// SIMATIC STEP 7 (V5.x) project CovesCAO
// CPU: CPU 315-2 PN/DP
// station: Hardware
// station: P_ADR_BUS
// station: Line04
// program: Engineering ZE25 - Common Program (Engineering) for Lines 01 & 02

SYMBOL_TABLE
"DB_GlobalData"	DB 1	DB 1	// Database global data
"DB_Keys"	DB 3	DB 3	// DB_Keys
"DB_Horn"	DB 5	DB 5	// Database Faults Horn request
"DB_VisuPara"	DB 6	DB 6	// Data from/to Visualizaton Parameter
"DB_VisuFaults"	DB 9	DB 9	// Data from/to Visualization Faults
"DB_VisuFaultsPrio"	DB 10	DB 10
"DB_CommWM001"	DB 40	DB 40	// DB_CommWM001
"DB_CommWM009"	DB 41	DB 41	// DB_CommWM009
"DB_CommWM011"	DB 42	DB 42	// DB_CommWM011
"DB_CommM0001"	DB 45	DB 45	// ABB ACS880 RPBA-01 interface EU MainDrive
"DB_CommM1103"	DB 46	DB 46	// ABB ACS880 RPBA-01 interface DT Sidefeeder
"DB_CommM0101"	DB 47	DB 47	// ABB ACS880 RPBA-01 interface BE BDP Dosing
"DB_CommM0102"	DB 48	DB 48	// ABB ACS880 RPBA-01 interface GR Pelletizer
"IDB_FB0"	DB 100	FB 0	// Instance data block of FB0
"IDB_FB1"	DB 101	FB 1	// Instance data block of FB1
"IDB_FB3"	DB 103	FB 3	// Instance data block of FB3
"IDB_FB4"	DB 104	FB 4	// Instance data block of FB4
"IDB_FB5"	DB 105	FB 5	// Instance data block of FB5
"IDB_FB6"	DB 106	FB 6	// Instance data block of FB6
"IDB_FB10"	DB 110	FB 10	// Instance data block of FB10
"IDB_FB11"	DB 111	FB 11	// Instance data block of FB11
"IDB_FB12"	DB 112	FB 12	// Instance data block of FB12
"IDB_FB13"	DB 113	FB 13	// Instance data block of FB13
"IDB_FB14"	DB 114	FB 14	// Instance data block of FB14
"IDB_FB15"	DB 115	FB 15	// Instance data block of FB15
"IDB_FB16"	DB 116	FB 16	// Instance data block of FB16
"IDB_FB17"	DB 117	FB 17	// Instance data block of FB17
"IDB_FB27"	DB 127	FB 27	// Instance data block of FB27
"IDB_FB28"	DB 128	FB 28	// Instance data block of FB28
"IDB_FB29"	DB 129	FB 29	// Instance data block of FB29
"IDB_FB30"	DB 130	FB 30	// Instance data block of FB30
"IDB_FB37"	DB 137	FB 37	// Instance data block of FB37
"IDB_FB40"	DB 140	FB 40	// Instance data block of FB40
"IDB_FB41"	DB 141	FB 41	// Instance data block of FB41
"IDB_FB42"	DB 142	FB 42	// Instance data block of FB42
"IDB_FB43"	DB 143	FB 43	// Instance data block of FB43
"IDB_FB44"	DB 144	FB 44	// Instance data block of FB44
"IDB_FB45"	DB 145	FB 45	// Instance data block of FB45
"IDB_FB46"	DB 146	FB 46	// Instance data block of FB46
"IDB_FB48"	DB 148	FB 48	// Instance data block of FB48
"IDB_FB49"	DB 149	FB 49	// Instance data block of FB49
"IDB_FB60"	DB 160	FB 60	// Instance data block of FB60
"IDB_FB61"	DB 161	FB 61	// Instance data block of FB61
"IDB_FB62"	DB 162	FB 62	// Instance data block of FB62
"IDB_FB70"	DB 170	FB 70	// Instance data block of FB70
"IDB_FB71"	DB 171	FB 71	// Instance data block of FB71
"IDB_FB72"	DB 172	FB 72	// Instance data block of FB72
"IDB_FB73"	DB 173	FB 73	// Instance data block of FB73
"IDB_FB74"	DB 174	FB 74	// Instance data block of FB74
"IDB_FB75"	DB 175	FB 75	// Instance data block of FB75
"IDB_FB76"	DB 176	FB 76	// Instance data block of FB76
"IDB_FB78"	DB 178	FB 78	// Instance data block of FB78
"IDB_FB100"	DB 1100	FB 100	// Instance data block of FB100
"IDB_FB112"	DB 1112	FB 112	// Instance data block of FB112
"IDB_FB116"	DB 1116	FB 116	// Instance data block of FB116
"IDB_FB117"	DB 1117	FB 117	// Instance data block of FB117
"Gen_Global"	FB 0	FB 0	// General Global
"Gen_GlobSig"	FB 1	FB 1	// General Global Signals
"EPGlobal"	FB 2	FB 2	// EPGlobal
"DPSlaveDiag"	FB 3	FB 3	// DP-Slave Diagnose
"FaultPrioSearch"	FB 4	FB 4	// MRoe Fault Priority Search
"HWButtonsStatus"	FB 5	FB 5	// HWButtonsStatus
"OperatingModes"	FB 6	FB 6	// OperatingModes Production / Maintenance
"BE_Org_Dos"	FB 10	FB 10	// BE Organisation Dosing
"BE_BC001DischargeFlap"	FB 11	FB 11	// BE BC001 discharge flap
"BE_BC001HopperInPos"	FB 12	FB 12	// BE BC001 hopper in position
"BE_BC001HopperPipeConn"	FB 13	FB 13	// BE BC001 hopper pipe connected
"BE_BC009DischargeAid"	FB 14	FB 14	// BE BC009 hopper discharge aid
"BE_BC009 DischargeFlap"	FB 15	FB 15	// BE_BC009 DischargeFlap
"BE_BC009 HopperInPos"	FB 16	FB 16	// BE_BC009 Hopper In Position
"BE_BC009HopperPipeConn"	FB 17	FB 17	// BE_BC009Hopper Pipe Connected
"BE_PA013Dosing"	FB 27	FB 27	// BE_PA013 dosing
"BE_PID PA013 OB35"	FB 28	FB 28	// BE PID controller for flow and temperature PA013 (OB35)
"BE_PA013Temperatures"	FB 29	FB 29	// BE_PA013Temperatures
"BE_PA013PropValve"	FB 30	FB 30	// PA013 proportional valve
"DT_EA011 Sidefeeder"	FB 37	FB 37	// DT EA011 Sidefeeder
"EU_Org_Extruder"	FB 40	FB 40	// EU Organisation Extruder - U0020
"EU_MainDrive"	FB 41	FB 41	// EU Extruder Main Drive - U0031
"EU_CoolingUnit"	FB 42	FB 42	// EU Cooling Unit - U0011
"EU_Clutch"	FB 43	FB 43	// EU extruder clutch
"EU_DriveCooling"	FB 44	FB 44	// EU main drive cooling - U0032
"EU_PIDCoolWaterTemp OB35"	FB 45	FB 45	// EU PID controller cooling water temperature (OB35)
"EU_NitrogenValve"	FB 46	FB 46	// EU Nitrogen valve
"EU_MeltPressTemp"	FB 48	FB 48	// EU extruder melt pressure and temperature
"EU_VacuumUnit"	FB 49	FB 49	// EU Extruder Vacuum Unit - U0024
"EU_Org_Heating"	FB 60	FB 60	// EU Organisation Heating
"EU_HeatingZone1"	FB 61	FB 61	// EU extruder heating zone 1 (feed zone)
"EU_HeatingZones2-11 OB35"	FB 62	FB 62	// EU Extruder Heating Zones 2 - 11 (OB35)
"GR_Org_Pel"	FB 70	FB 70	// GR Organisation Pelletizer
"GR_WaterBath"	FB 71	FB 71	// GR water bath pump - U0021
"GR_Dewatering"	FB 72	FB 72	// GR drive fan strand dewatering - U0022
"GR_Classifier"	FB 73	FB 73	// GR Classifier
"GR_SafetyKey"	FB 74	FB 74	// GR safety key
"GR_Pelletizer"	FB 75	FB 75	// GR pelletizer - U0023
"GR_PIDWaterBath"	FB 76	FB 76	// GR Water bath
"GR_DownstTotalizer"	FB 78	FB 78	// GR_DownstTotalizer
"DT_Org_Dos"	FB 100	FB 100	// DT Organisation Dosierung
"DT_WM001"	FB 112	FB 112	// DT WM001Brabender
"DT_WM009"	FB 116	FB 116	// DT WM009 KTron
"DT_WM011"	FB 117	FB 117	// DT_WM011 K-Tron
"EPTimerOn"	FB 304	FB 304
"EPTimerOff"	FB 305	FB 305
"EPSetDateTime"	FB 307	FB 307	// Set Date and Time by UDT0
"EPFindMaxDINT"	FB 309	FB 309	// EPFindMaxDINT
"EPFilter"	FB 311	FB 311
"EPExPulsGen"	FB 317	FB 317	// EPExPulsGen
"EPThermIntegLoss"	FB 318	FB 318
"EPTempRamp"	FB 319	FB 319
"EPAverageVari"	FB 323	FB 323
"EPMotorN1FB"	FB 325	FB 325
"EPValveNC"	FB 336	FB 336	// EPValveNC
"EPFault"	FB 341	FB 341	// EPFault
"EPPreHeatTime"	FB 357	FB 357	// Extruder control and converting the pre heating time
"EPLevelSwitch"	FB 376	FB 376
"EPActValue"	FB 386	FB 386	// handling of ActREAL (modular SPS-datatype)
"EPRunTimeMeter"	FB 391	FB 391
"EPTotalPulse"	FB 392	FB 392
"EPToggle8"	FB 397	FB 397	// EPToggle8
"EPTcontZone"	FB 427	FB 427	// Extruder heating zone of tcont cp
"CONT_C"	FB 541	FB 541	// Continuous Control
"PULSEGEN"	FB 543	FB 543	// Pulse Generation
"TCONT_CP"	FB 558	FB 558	// temperature PID controller with pulse generator and self-tuning
"FCStatusWordsToVisu"	FB 603	FB 603	// FCStatusWordsToVisu
"BAYERDeviationAlmWarn"	FB 604	FB 604	// BAYERDeviationAlmWarn
"RF_RampAutoPush"	FB 615	FB 615	// Ramp value automatic to OP or inc/dec value by switches
"MR_TempZoneSimple"	FB 616	FB 616	// MR_TempZoneSimple
"CTBDHFlt"	FB 1000	FB 1000	// Störung für Dosierer
"CTKDLFlt"	FB 1001	FB 1001	// Dosierer K-Tron Detailstörungen
"EPGraph10Pos"	FB 1219	FB 1219
"EPRampOP_neu"	FB 1269	FB 1269	// EPRampOP_neu
"EPNomFilter"	FB 1270	FB 1270	// filtering of a nominal REAL value
"EPLocalMode"	FB 1282	FB 1282	// EPLocalMode
"EPTimerOn_neu"	FB 1304	FB 1304	// EPTimerOn_neu
"EPTimerOff_neu"	FB 1305	FB 1305	// EPTimerOff_neu
"EPAverageVari_Neu"	FB 1323	FB 1323
"EPMsg"	FB 1341	FB 1341
"EPSlaveDiagDP"	FB 1346	FB 1346	// Slave Diag DP
"EPToggel8_neu"	FB 1397	FB 1397	// EPToggel8_neu
"EP MS DataChange REAL"	FB 1501	FB 1501	// master - slave datachange handler for REAL values
"EP MS DataChange BOOL"	FB 1502	FB 1502	// master - slave datachange handler for boolean signals
"EP Comm ISC-CM Plus"	FB 1530	FB 1530	// Comm ISC-CM Plus
"EP ISC-CMp H Feeder"	FB 1535	FB 1535	// Brabender ISC CM plus H-type dosing feeder
"EP Comm K-Link KCM / SCM"	FB 1540	FB 1540	// Communication to K-Tron Smart K-Link KCM or SCM
"CT KCM LWF Feeder"	FB 1545	FB 1545	// K-Tron Smart K-Link KCM LWF-type dosing feeder
"GE_DT"	FC 12	FC 12	// Greater or Equal DT
"GT_DT"	FC 14	FC 14	// Greater Than DT
"SB_DT_TM"	FC 35	FC 35	// Subtract DT Time
"EPOperationMessage"	FC 301	FC 301	// Block vor one operation message
"EPNomLight"	FC 302	FC 302	// EPNomLight
"EPStartStop"	FC 307	FC 307	// EPStartStop
"EPToggle1"	FC 309	FC 309	// EPToggle1
"EPLimitAlarmReal"	FC 320	FC 320	// limit alarm generation
"EPAnyBitSet"	FC 349	FC 349	// EPAnyBitSet
"EPAnalogInReal"	FC 351	FC 351	// EPAnalogInReal
"EPAnalogOutReal"	FC 361	FC 361	// EPAnalogOutReal
"EPNominalComponent"	FC 365	FC 365	// nominal calculation of one dosing component
"EPMinuteImpulse"	FC 383	FC 383	// EPMinuteImpulse
"BAYERNomLightStartup"	FC 502	FC 502	// BAYERNomLight with Startup value handling
"EPNomLightDINT"	FC 503	FC 503	// EPNomLightDINT
"EPBAYER_TSD"	FC 505	FC 505	// EPBAYER Theoretical Strand Diameter
"EPBAYER_UPOStat"	FC 506	FC 506	// EPBAYER_UPOStat
"ClearBitsDelayed"	FC 510	FC 510	// ClearBitsDelayed
"EPGraphCalc"	FC 1219	FC 1219	// GraphCalc
"EPStatText"	FC 1300	FC 1300	// EP Status Text
"EPStat"	FC 1301	FC 1301	// common Status for Visu
"=PS230+SK02-1F4:14"	I 0.0	BOOL	// CIRCUIT BREAKER 230VAC O.K.
"=PS24+SK02-2F5:14"	I 0.1	BOOL	// CIRCUIT BREAKER 24VDC CONTROL VOLTAGE O.K.
"=PS24+SK02-3F5:14"	I 0.2	BOOL	// CIRCUIT BREAKER 24VDC LOAD VOLTAGE O.K.
"=ES+SK02-2K3:94"	I 0.3	BOOL	// EMERGENCY STOP RELAY ON
"=ES+CP01-3S1:34"	I 0.4	BOOL	// EMERGENCY STOP CONTROL PANEL EXTRUDER
"=ES+CP02-3S2:32"	I 0.5	BOOL	// NOT EMERGENCY STOP CONTROL PANEL PELLETIZER
"=ES+CP03-3S3:34"	I 0.6	BOOL	// EMERGENCY STOP EXTERNAL
"=ES+CP04-3S4:34"	I 0.7	BOOL	// EMERGENCY STOP EXTERNAL
"=EU04+CP01-1S1:14"	I 1.0	BOOL	// LAMP TEST
"=EU04+CP01-1S2:14"	I 1.1	BOOL	// HORN OFF
"=EU04+CP01-1S3:14"	I 1.2	BOOL	// H0008 AUXILIARY DRIVES START
"=EU04+CP01-1S4:12"	I 1.3	BOOL	// H0008 AUXILIARY DRIVES STOP
"=EU04+CP01-1S5:14"	I 1.4	BOOL	// H0001 EXTRUDER MAIN DRIVE START
"=EU04+CP01-1S6:12"	I 1.5	BOOL	// H0001 EXTRUDER MAIN DRIVE STOP
"=EU04+CP01-1S7:24"	I 1.6	BOOL	// H0009 EXTRUDER -
"=EU04+CP01-1S7:14"	I 1.7	BOOL	// H0009 EXTRUDER +
"=EU04+CP01-2S1:14"	I 2.0	BOOL	// H0101 FEEDING SYSTEM START
"=EU04+CP01-2S2:12"	I 2.1	BOOL	// H0101 FEEDING SYSTEM STOP
"=EU04+CP01-2S3:24"	I 2.2	BOOL	// H0102 FEEDING -
"=EU04+CP01-2S3:14"	I 2.3	BOOL	// H0102 FEEDING +
"+CP01-X4:14"	I 2.4	BOOL	// SPARE
"+CP01-X4:15"	I 2.5	BOOL	// SPARE
"+CP01-X4:16"	I 2.6	BOOL	// SPARE
"=ILUM+CP01-1E1:5"	I 2.7	BOOL	// COOLING UNIT CABINET +CP01 OK
"=GR04+CP02-1S4:24"	I 3.0	BOOL	// CUTTER SLOW
"=GR04+CP02-1S2:14"	I 3.1	BOOL	// CUTTER SRART
"=GR04+CP02-1S1:12"	I 3.2	BOOL	// CUTTER STOP
"=GR04+CP02-1S3:14"	I 3.3	BOOL	// LOCAL
"=GR04+CP02-1S3:24"	I 3.4	BOOL	// REMOTE
"=GR04+CP02-1S4:14"	I 3.5	BOOL	// CUTTER FAST
"=GR04+CP02-1S5:22"	I 3.6	BOOL	// FEED ROLL UP PRESSURE ON
"=GR04+CP02-1S5:14"	I 3.7	BOOL	// FEED ROLL UP PRESSURE OFF
"=BE04+BC001-G0014:4"	I 4.0	BOOL	// HOPPER BC001 IN POSITION
"=BE04+XB001-G0013:BK"	I 4.1	BOOL	// XB001 DISCHARGE PIPE CONNECTED
"=BE04+BC009-G0094:4"	I 4.2	BOOL	// HOPPER BC009 IN POSITION
"=DT04+WM001-H0101:14"	I 4.3	BOOL	// EXTRUDER DOSING WM001 MAINTENANCE SWITCH ON
"=BE04+XB009-G0093:BK"	I 4.4	BOOL	// XB009 DISCHARGE PIPE CONNECTED
"I4.5"	I 4.5	BOOL	// SPARE
"I4.6"	I 4.6	BOOL	// SPARE
"=DT04+WM011-M1101:J5:5"	I 4.7	BOOL	// DOSING UNIT WM011 REFILL
"=DT04+WM011-H1101:6"	I 5.0	BOOL	// DOSING UNIT WM011 MAINTENANCE SWITCH ON
"=DT04+WM009-M0901:J5:5"	I 5.1	BOOL	// DOSING UNIT WM009 REFILL
"=DT04+WM009-H0901:6"	I 5.2	BOOL	// DOSING UNIT WM009 MAINTENANCE SWITCH ON
"=ES+SK02-2K1:X2:Y32"	I 5.3	BOOL	// EMERGENCY STOP OK
"=ES+CP01-1S1:14"	I 5.4	BOOL	// LOAD VOLTAGE ON
"=DT04+WM009-G0901:WH"	I 5.5	BOOL	// DOSING UNIT WM009 SAFETY SWITCH
"I5.6"	I 5.6	BOOL	// SPARE
"I5.7"	I 5.7	BOOL	// SPARE
"I8.0"	I 8.0	BOOL	// SPARE
"I8.1"	I 8.1	BOOL	// SPARE
"=EU04+GA001-G0001:BK"	I 8.2	BOOL	// CLUTCH CONTROL
"I8.3"	I 8.3	BOOL	// SPARE
"I8.4"	I 8.4	BOOL	// SPARE
"I8.5"	I 8.5	BOOL	// SPARE
"=EU04+SK02-8Q1:14"	I 8.6	BOOL	// PUMP TEMPERING UNIT EXTRUDER MOTOR PROTECT. O.K.
"=EU04+PA001-H0011:14"	I 8.7	BOOL	// PUMP TEMPERING UNIT MAINTENANCE SWITCH ON
"=EU04+BA001-L0011:BK"	I 10.0	BOOL	// COOLING WATER HIGH
"=EU04+BA001-L0011:GY"	I 10.1	BOOL	// COOLING WATER NOT LOW
"+SK02-X4:97"	I 10.2	BOOL	// SPARE
"=EU04+SK02-40K1:X2:Y32"	I 10.3	BOOL	// EXTRUDER SAFETY SWITCH OK
"=EU04+GA001-G0002:8"	I 10.4	BOOL	// SAFETY SWITCH OF CONNECTION PART COVER LEFT
"=EU04+GA001-G0003:8"	I 10.5	BOOL	// SAFETY SWITCH OF CONNECTION PART COVER RIGHT
"=EU04+GA001-G0004:8"	I 10.6	BOOL	// SAFETY SWITCH OF COUPLING COVER
"=EU04+GA001-G0005:8"	I 10.7	BOOL	// SAFETY SWITCH HOPPER COVER
"=EU04+GA001-F0041:4"	I 11.0	BOOL	// EXTRUDER NITROGEN FLOW SWITCHING POINT A
"=EU04+GA001-F0041:2"	I 11.1	BOOL	// EXTRUDER NITROGEN FLOW SWITCHING POINT B
"I11.2"	I 11.2	BOOL	// SPARE
"I11.3"	I 11.3	BOOL	// SPARE
"I11.4"	I 11.4	BOOL	// SPARE
"I11.5"	I 11.5	BOOL	// SPARE
"I11.6"	I 11.6	BOOL	// SPARE
"I11.7"	I 11.7	BOOL	// SPARE
"=EU04+SK02-13A1:2"	I 32.0	BOOL	// EXTRUDER ZONE 2 CURRENT CONTROL O.K.
"=EU04+SK02-15A1:2"	I 32.1	BOOL	// EXTRUDER ZONE 3 CURRENT CONTROL O.K.
"=EU04+SK02-17A1:2"	I 32.2	BOOL	// EXTRUDER ZONE 4 CURRENT CONTROL O.K.
"=EU04+SK02-19A1:2"	I 32.3	BOOL	// EXTRUDER ZONE 5 CURRENT CONTROL O.K.
"=EU04+SK02-21A1:2"	I 32.4	BOOL	// EXTRUDER ZONE 6 CURRENT CONTROL O.K.
"=EU04+SK02-23A1:2"	I 32.5	BOOL	// EXTRUDER ZONE 7 CURRENT CONTROL O.K.
"=EU04+SK02-25A1:2"	I 32.6	BOOL	// EXTRUDER ZONE 8 CURRENT CONTROL O.K.
"=DT04+EA011-H1103:14"	I 32.7	BOOL	// SIDE FEEDER MAINTENANCE SWITCH ON
"=EU04+SK02-29A1:2"	I 33.0	BOOL	// EXTRUDER ZONE 10 CURRENT CONTROL O.K.
"=DT04+EA011-H1104:14"	I 33.1	BOOL	// SIDE FEEDER VACUUMPUMP ON
"=EU04+SK02-32K1:X6:OU2"	I 33.2	BOOL	// EXTRUDER MELT PRESSURE NOT MAX MAX
"=EU04+SK02-32K1:X6:OU1"	I 33.3	BOOL	// DIFFERENTIAL PRESSURE P1.1 <--> P1.2 MAX MAX
"=EU04+SK02-33K1:X6:OU1"	I 33.4	BOOL	// EXTRUDER ZONE 8 MELT PRESSURE MAX. MAX.
"=DT04+SK02-11Q1:14"	I 33.5	BOOL	// SIDE FEEDER VACUUMPUMP MOTOR PROTECT. O.K.
"=EU04+SK02-31A1:2"	I 33.6	BOOL	// EXTRUDER ZONE 11 CURRENT CONTROL O.K.
"I33.7"	I 33.7	BOOL	// SPARE
"=EU04+SK01-10T1:8"	I 140.0	BOOL	// VACUUM UNIT SEPARATOR NOT EMPTY
"=BE04+SK01-4Q1:14"	I 140.1	BOOL	// PA013 PUMP DRIVE MOTOR PROTECTION OK
"=BE04+PA013-H0101:14"	I 140.2	BOOL	// PUMP DRIVE PA013 MAINTENANCE SWITCH ON
"=BE04+SK01-8A1:12"	I 140.3	BOOL	// PA013 HEATER PUMP ZONE 2 CURRENT CONTROL O.K.
"=BE04+PA013-P0101:2"	I 140.4	BOOL	// PA013 PRESSURE >MIN
"I140.5"	I 140.5	BOOL	// SPARE
"=BE04+PA013-G0102:2"	I 140.6	BOOL	// PA013 GATE VALVE TO EXTRUDER OPEN
"=BE04+PA013-G0102:3"	I 140.7	BOOL	// PA013 GATE VALVE TO EXTRUDER CLOSED
"=BE04+PA013-G0101:2"	I 141.0	BOOL	// PA013 GATE VALVE RETURN FLOW OPENED
"=BE04+PA013-G0101:3"	I 141.1	BOOL	// PA013 GATE VALVE RETURN FLOW CLOSED
"=GR04+SK01-21Q1:14"	I 141.2	BOOL	// CLASSIFIER VIBRATOR MOTOR PROTECTION OK
"=EU04+SK01-11T1:12"	I 141.3	BOOL	// VACUUM UNIT SEPARATOR TEMPERATURE WARNING
"=GR04+SK01-13K1:Y32"	I 141.4	BOOL	// PELLETIZER NOT RUNNING
"=GR04+SK01-13K1:Y35"	I 141.5	BOOL	// PELLETIZER FAULT
"=EU04+GM001-H0001:14"	I 141.6	BOOL	// EXTRUDER DRIVE MAINTENANCE SWITCH ON
"=GR04+SK01-11Q1:14"	I 141.7	BOOL	// PELLETIZER DRIVE MOTOR PROTECTION OK
"=EU04+VP001-H0201:14"	I 142.0	BOOL	// VACUUM PUMP EXTRUDER MAINTENANCE SWITCH ON
"=EU04+SK01-8Q1:14"	I 142.1	BOOL	// VACUUM PUMP EXTRUDER MOTOR PROTECT. O.K.
"=GR04+PA001-H0201:14"	I 142.2	BOOL	// PUMP WATER BATH MAINTENANCE SWITCH ON
"I142.3"	I 142.3	BOOL	// SPARE
"I142.4"	I 142.4	BOOL	// SPARE
"=GR04+SK01-11Q2:14"	I 142.5	BOOL	// PELLETIZER DRIVE MOTOR CONTACTOR ON FEEDBACK MONITORING
"=ILUM+SK01-3E1:X1"	I 142.6	BOOL	// AIR CONDITIONER NO FAULT
"=GR04+ZA001-G0030:5"	I 142.7	BOOL	// SAFETY DOOR CLOSED
"=GR04+SK01-1Q1:14"	I 143.0	BOOL	// PUMP WATER BATH MOTOR PROTECT. O.K.
"I143.1"	I 143.1	BOOL	// SPARE
"I143.2"	I 143.2	BOOL	// SPARE
"=GR04+SK01-15K1:X2:Y32"	I 143.3	BOOL	// PELLETIZER KEY PLUGGED
"=ML04+PM001-SE-K1"	I 143.4	BOOL	// PACKING MACHINE RUNNING
"=ML04+PM001-SE-K2"	I 143.5	BOOL	// PACKING MACHINE FAULT
"=ML04+PM001-SE-K3"	I 143.6	BOOL	// PACKING MACHINE CONVEYOR RUNNING
"=ML04+PM001-SE-K4"	I 143.7	BOOL	// PACKING MACHINE BAG COUNTER
"=EU04+VP001-P0083:4"	I 144.0	BOOL	// VACUUM UNIT PRESSURE INDICATOR
"=EU04+SK01-12T1:21"	I 144.1	BOOL	// VACUUM UNIT FLOW SWITCH MIN
"=EU04+SK01-12T1:17"	I 144.2	BOOL	// VACUUM UNIT FLOW SWITCH FAULT
"=EU04+SK01-7Q1:14"	I 144.3	BOOL	// EXTRUDER FREMDBELÜFTUNG MOTOR PROTECT. O.K.
"+SK01-X7:37"	I 144.4	BOOL	// SPARE
"=DT04+SK01-1Q1:14"	I 144.5	BOOL	// SIDE FEEDER MOTOR PROTECT. O.K.
"+SK01-X7:38"	I 144.6	BOOL	// SPARE
"=EU04+GM001-H0002:14"	I 144.7	BOOL	// EXTRUDER FREMDBELÜFTUNG MAINTENANCE SWITCH ON
"Clock10000mHz"	M 0.0	BOOL	// clock signal 10Hz / 100ms
"Clock5000mHz"	M 0.1	BOOL	// clock signal 5Hz / 200ms
"Clock2500mHz"	M 0.2	BOOL	// clock signal 2,5Hz / 400ms
"Clock2000mHz"	M 0.3	BOOL	// clock signal 2Hz / 500ms
"Clock1250mHz"	M 0.4	BOOL	// clock signal 1,25Hz / 800ms
"Clock1000mHz"	M 0.5	BOOL	// clock signal 1Hz / 1s
"Clock625mHz"	M 0.6	BOOL	// clock signal 0,625Hz / 1,6s
"Clock500mHz"	M 0.7	BOOL	// clock signal 0,5Hz / 2s
"Impulse100ms"	M 1.0	BOOL	// impulse signal each 100ms
"Impulse200ms"	M 1.1	BOOL	// impulse signal each 200ms
"Impulse400ms"	M 1.2	BOOL	// impulse signal each 400ms
"Impulse500ms"	M 1.3	BOOL	// impulse signal each 500ms
"Impulse800ms"	M 1.4	BOOL	// impulse signal each 800ms
"Impulse1000ms"	M 1.5	BOOL	// impulse signal each 1000ms
"Impulse1600ms"	M 1.6	BOOL	// impulse signal each 1600ms
"Impulse2000ms"	M 1.7	BOOL	// impulse signal each 2000ms
"StartUpPLC"	M 2.0	BOOL	// start up signal, set in OB100/OB101/OB102, reset at end of program
"BatteryFault"	M 2.1	BOOL	// battery fault, set in OB81
"ControlVoltageOn"	M 2.2	BOOL	// control voltage on signal
"ControlVoltageOnDel"	M 2.3	BOOL	// control voltage on delayed signal
"LoadVoltageOn"	M 2.4	BOOL	// load voltage on signal extruder
"LoadVoltageOnDel"	M 2.5	BOOL	// load voltage on delayed signal extruder
"FaultAck"	M 2.6	BOOL	// fault acknowledge signal
"FaultAckExt"	M 2.7	BOOL	// fault acknowledge extended signal
"Impulse1min"	M 3.0	BOOL	// impulse signal each 1min
"LampTest"	M 3.1	BOOL	// extendet signal for lamp test
"BlockFault"	M 3.2	BOOL	// block fault signal
"HornAck"	M 3.3	BOOL	// horn acknowledge signal
"HornAckExt"	M 3.4	BOOL	// horn acknowledge extended signal
"ContrVoltageOnDel_Block"	M 3.5	BOOL	// block fault if control voltage is missing
"FaultAckOB35"	M 3.6	BOOL	// fault acknowledge signal for OB35
"HornAckOB35"	M 3.7	BOOL	// horn acknowledge signal for OB35
"LoadVoltageOnDel_Block"	M 4.0	BOOL	// block fault if load voltage is missing
"StartUpPLC_OB35"	M 4.4	BOOL	// start up signal for OB35, set in OB100/OB101/OB102, reset at end of OB35
"FaultOB80"	M 6.0	BOOL	// Fault: OB 80 called, cycle time error
"FaultOB81"	M 6.1	BOOL	// Fault: OB 81 called, power supply error
"FaultOB82"	M 6.2	BOOL	// Fault: OB 82 called, I/O point error 1
"FaultOB83"	M 6.3	BOOL	// Fault: OB 83 called, I/O point error 2
"FaultOB84"	M 6.4	BOOL	// Fault: OB 84 called, cpu error
"FaultOB85"	M 6.5	BOOL	// Fault: OB 85 called, OB not loaded
"FaultOB86"	M 6.6	BOOL	// Fault: OB 86 called, rack fault
"FaultOB87"	M 6.7	BOOL	// Fault: OB 87 called, communication fault
"FaultOB88"	M 7.0	BOOL	// Fault: OB 88 called, breakup error
"FaultOB121"	M 7.1	BOOL	// Fault: OB121 called, programming error
"FaultOB122"	M 7.2	BOOL	// Fault: OB122 called, module access error
"Simulation"	M 8.0	BOOL	// request start simulation [1=requested]
"IB_0"	M 10.0	BOOL	// commissioning & test always FALSE
"IB_1"	M 10.1	BOOL	// commissioning & test always TRUE
"IB_DummyOut"	M 10.2	BOOL	// commissioning & test for dummy outputs
"Alarm_Prio1"	M 100.0	BOOL	// Alarm with Priority 1 - safety alarm
"Alarm_Prio2"	M 100.1	BOOL	// Alarm with Priority 2 - process related alarm with interlock
"Alarm_Prio3"	M 100.2	BOOL	// Alarm with Priority 3 - process related alarm without interlock
"Alarm_Prio4"	M 100.3	BOOL	// Alarm with Priority 4 - event
"Alarm_Prio5"	M 100.4	BOOL	// Alarm with Priority 5 - system alarm
"FlagImpCoolDownOff"	M 110.2	BOOL	// Flag Impuls CoolDown Function Off
"ImpPA013PelletizerOff"	M 110.5	BOOL	// Impuls Pelletizer delayed off after PA013 Stop
"FlagImpPA013PelletOff"	M 111.5	BOOL	// Flag Impuls Pelletizer delayed off after PA013 Stop
"ClockByte"	MB 0	BYTE	// byte for clock signals
"ImpulseByte"	MB 1	BYTE	// byte for impulses
"MD10"	MD 10	REAL	// commissioning & test
"CycleExecution"	OB 1	OB 1	// CycleExecution
"CYC_INT5"	OB 35	OB 35	// Cyclic Interrupt 3
"CYCL_FLT"	OB 80	OB 80	// Cycle Time Fault
"I/O_FLT1"	OB 82	OB 82	// I/O Point Fault 1
"I/O_FLT2"	OB 83	OB 83	// I/O Point Fault 2
"OBNL_FLT"	OB 85	OB 85	// OB Not Loaded Fault
"RACK_FLT"	OB 86	OB 86	// Loss of Rack Fault
"COMM_FLT"	OB 87	OB 87	// Communication Fault
"EPCompleteRestart"	OB 100	OB 100	// EPCompleteRestart
"PROG_ERR"	OB 121	OB 121	// Programming Error
"MOD_ERR"	OB 122	OB 122	// Module Access Error
"=EU04+EA001-T0003:Fe"	PIW 320	INT	// EXTRUDER FEED ZONE TEMPERATURE
"=EU04+EA001-T0021:Fe"	PIW 322	INT	// EXTRUDER ZONE 2 TEMPERATURE
"=EU04+EA001-T0031:Fe"	PIW 324	INT	// EXTRUDER ZONE 3 TEMPERATURE
"=EU04+EA001-T0041:Fe"	PIW 326	INT	// EXTRUDER ZONE 4 TEMPERATURE
"=EU04+EA001-T0051:Fe"	PIW 328	INT	// EXTRUDER ZONE 5 TEMPERATURE
"=EU04+EA001-T0061:Fe"	PIW 330	INT	// EXTRUDER ZONE 6 TEMPERATURE
"=EU04+EA001-T0071:Fe"	PIW 332	INT	// EXTRUDER ZONE 7 TEMPERATURE
"=EU04+EA001-T0081:Fe"	PIW 334	INT	// EXTRUDER ZONE 8 TEMPERATURE
"PIW336"	PIW 336	INT	// SPARE
"PIW338"	PIW 338	INT	// SPARE
"=EU04+EA001-T0101:Fe"	PIW 340	INT	// EXTRUDER ZONE 10 TEMPERATURE
"=EU04+EA001-T0102:Fe"	PIW 342	INT	// EXTRUDER ZONE 11 TEMPERATURE
"=EU04+EA001-T0112:Fe"	PIW 344	INT	// EXTRUDER MELT TEMPERATURE
"=EU04+PA001-T0011:Fe"	PIW 346	INT	// TEMPERATURE COOLING WATER TEMPERING UNIT
"PIW348"	PIW 348	INT	// SPARE
"PIW350"	PIW 350	INT	// SPARE
"=EU04+SK02-32K1:X4:1"	PIW 352	INT	// MELT PRESSURE P1.1 ACTUAL VALUE
"=EU04+SK02-32K1:X4:2"	PIW 354	INT	// MELT PRESSURE P1.2 ACTUAL VALUE
"=EU04+SK02-33K1:X4:1"	PIW 356	INT	// EXTRUDER MELT PRESSURE ACTUAL VALUE
"=EU04+GA001-F0041:5"	PIW 358	INT	// EXTRUDER NITROGEN FLOW ACTUAL VALUE
"=BE04+BC001-Y0012:9"	PIW 360	INT	// DISCHARGE FLAP BC001 OPEN ACTUAL VALUE
"PIW362"	PIW 362	INT	// SPARE
"=BE04+BC009-Y0092:9"	PIW 364	INT	// DISCHARGE FLAP BC009 OPEN ACTUAL VALUE
"PIW366"	PIW 366	INT	// SPARE
"PIW368"	PIW 368	INT	// SPARE
"PIW370"	PIW 370	INT	// SPARE
"PIW372"	PIW 372	INT	// SPARE
"PIW374"	PIW 374	INT	// SPARE
"=BE04+PA013-T0313:1"	PIW 380	INT	// PA013 TEMPERATURE ZONE 1 BEVORE PUMPE
"=BE04+PA013-T0314:1"	PIW 382	INT	// PA013 TEMPERATURE ZONE 3 PUMP
"=BE04+PA013-T0315:1"	PIW 384	INT	// PA013 TEMPERATURE ZONE 4 AFTER PUMP
"=BE04+PA013-T0316:1"	PIW 386	INT	// PA013 TEMPERATURE ZONE 5 ANSCHLUSSSTÜCK EXTRUDER
"=BE04+PA013-T0102:1"	PIW 388	INT	// PA013 TEMPERATURE PUMP ZONE 2
"=GR04+FB001-T0042:1"	PIW 390	INT	// CLASSIFIER FB001 TEMPERATURE PRODUCT
"=BE04+PA013-T0107:1"	PIW 392	INT	// PA013 TEMPERATURE PRODUCT
"PIW394"	PIW 394	INT	// SPARE
"+SK01-X7:39"	PIW 396	INT	// SPARE
"=EU04+VP001-P0083:2"	PIW 398	INT	// VACUUM UNIT ACTUAL PRESSURE
"=GR04+WX001-T0011:+"	PIW 400	INT	// RECIRCLE WATER SUPPLY TEMPERATURE
"=GR04+WX001-T0012:+"	PIW 402	INT	// RECIRCLE WATER RETURE TEMPERATURE
"=EU04+SK01-11T1:7"	PIW 404	INT	// VACUUM UNIT SEPARATOR TEMPERATURE ACTUAL VALUE
"=GR04+FA001-P0101:1"	PIW 406	INT	// COOLING WATER PRESSURE ACTUAL VALUE
"=BE04+PA013-F0101:26"	PIW 408	INT	// PA013 FLOW MEASURING ACTUAL VALUE
"=BE04+PA013-P0102:1"	PIW 410	INT	// PA013 BDP DOSING PRESSURE ACTUAL VALUE
"=BE04+BC001-Y0012:1"	PQW 320	INT	// DISCHARGE FLAP BC001 OPEN NOMINAL VALUE
"=BE04+BC009-Y0092:1"	PQW 322	INT	// DISCHARGE FLAP BC009 OPEN NOMINAL VALUE
"PQW324"	PQW 324	INT	// SPARE
"PQW326"	PQW 326	INT	// SPARE
"=BE04+PA013-Y1320:11"	PQW 380	INT	// PA013 PROPORTIONAL VALVE
"=GR04+WA001-Y0011:11"	PQW 382	INT	// COOLING WATER RETURN VALVE
"PQW336"	PQW 384	INT	// SPARE
"PQW338"	PQW 386	INT	// SPARE
"=EU04+CP01-3P2:X1"	Q 0.0	BOOL	// LOAD VOLTAGE ON
"=EU04+CP01-3P3:X1"	Q 0.1	BOOL	// X0008 AUXILIARY DRIVES ON
"=EU04+CP01-3P4:X1"	Q 0.2	BOOL	// X0001 EXTRUDER MAIN DRIVE ON
"=EU04+CP01-3P5:X1"	Q 0.3	BOOL	// X0101 FEEDING SYSTEM ON
"+CP01-X4:25"	Q 0.4	BOOL	// SPARE
"+CP01-X4:26"	Q 0.5	BOOL	// SPARE
"+CP01-X4:27"	Q 0.6	BOOL	// SPARE
"+CP01-X4:28"	Q 0.7	BOOL	// SPARE
"Q1.0"	Q 1.0	BOOL	// SPARE
"Q1.1"	Q 1.1	BOOL	// SPARE
"Q1.2"	Q 1.2	BOOL	// SPARE
"=EU04+SK02-40K2:A1"	Q 1.3	BOOL	// EXTRUDER SAFETY SWITCH RESET
"Q1.4"	Q 1.4	BOOL	// SPARE
"=GR04+CP02-2P3:X1"	Q 1.5	BOOL	// CUTTER INTERLOCKING SYSTEM RELEASE
"=GR04+CP02-2P1:X1"	Q 1.6	BOOL	// CUTTER ON
"=GR04+CP02-2P2:X1"	Q 1.7	BOOL	// FEED ROLL UP PRESSURE OFF
"=DT04+WM001-2A2:68"	Q 2.0	BOOL	// DOSING UNIT WM001 RELEASE
"=DT04+SK02-8K1:A1"	Q 2.1	BOOL	// DOSING UNIT WM011 INTERLOCKING ON
"=DT04+SK02-6K1:A1"	Q 2.2	BOOL	// DOSING UNIT WM009 INTERLOCKING ON
"=ES+SK02-1K1:A1"	Q 2.3	BOOL	// EMERGENCY STOP RESET
"Q2.4"	Q 2.4	BOOL	// SPARE
"Q2.5"	Q 2.5	BOOL	// SPARE
"Q2.6"	Q 2.6	BOOL	// SPARE
"Q2.7"	Q 2.7	BOOL	// SPARE
"Q 3.0"	Q 3.0	BOOL	// spare
"=EU04+GA001-Y0012"	Q 3.1	BOOL	// COOLING WATER EXTRUDER GEAR BOX OPEN
"=EU04+SK02-8Q2:A1"	Q 3.2	BOOL	// PUMP TEMPERING UNIT EXTRUDER ON
"=EU04+WA001-Y0012:A1"	Q 3.3	BOOL	// COOLING WATER TEMPERING UNIT OPEN
"Q3.4"	Q 3.4	BOOL	// SPARE
"Q3.5"	Q 3.5	BOOL	// SPARE
"Q3.6"	Q 3.6	BOOL	// SPARE
"=EU04+BA001-Y0011:A1"	Q 3.7	BOOL	// INLET COOLING WATER TEMPERING UNIT OPEN
"=EU04+SK02-13V1:A1"	Q 32.0	BOOL	// EXTRUDER ZONE 2 HEATING ON
"=EU04+SK02-15V1:A1"	Q 32.1	BOOL	// EXTRUDER ZONE 3 HEATING ON
"=EU04+SK02-17V1:A1"	Q 32.2	BOOL	// EXTRUDER ZONE 4 HEATING ON
"=EU04+SK02-19V1:A1"	Q 32.3	BOOL	// EXTRUDER ZONE 5 HEATING ON
"=EU04+SK02-21V1:A1"	Q 32.4	BOOL	// EXTRUDER ZONE 6 HEATING ON
"=EU04+SK02-23V1:A1"	Q 32.5	BOOL	// EXTRUDER ZONE 7 HEATING ON
"=EU04+SK02-25V1:A1"	Q 32.6	BOOL	// EXTRUDER ZONE 8 HEATING ON
"=EU04+GA001-Y0045:1"	Q 32.7	BOOL	// EXTRUDER NITROGEN VALVE
"=EU04+SK02-29V1:A1"	Q 33.0	BOOL	// EXTRUDER ZONE 10 HEATING ON
"=EU04+SK02-31V1:A1"	Q 33.1	BOOL	// EXTRUDER ZONE 11 HEATING ON
"Q33.2"	Q 33.2	BOOL	// SPARE
"=BE04+BC009-Y0093:1"	Q 33.3	BOOL	// HOPPER BC009 KNOCKER ON
"=DT04+VP011-Y1101:1"	Q 33.4	BOOL	// SIDE FEEDER VACUUMPUMP AIR PURGE VALVE
"=DT04+VP011-Y1102:1"	Q 33.5	BOOL	// SIDE FEEDER VACUUMPUMP SUCTION VALVE
"=DT04+SK02-11Q2:A1"	Q 33.6	BOOL	// SIDE FEEDER VACUUMPUMP ON
"Q33.7"	Q 33.7	BOOL	// SPARE
"=EU04+SK02-32K1:X3:IN1"	Q 34.0	BOOL	// EXTRUDER MELT PRESSURE CALIBRATION
"=EU04+SK02-32K1:X3:IN3"	Q 34.1	BOOL	// EXTRUDER MELT PRESSURE RESET FAULT
"=EU04+SK02-33K1:X3:IN3"	Q 34.2	BOOL	// EXTRUDER MELT PRESSURE RESET FAULT
"=EU04+SK02-33K1:X3:IN1"	Q 34.3	BOOL	// EXTRUDER MELT PRESSURE CALIBRATION
"Q34.4"	Q 34.4	BOOL	// SPARE
"Q34.5"	Q 34.5	BOOL	// SPARE
"Q34.6"	Q 34.6	BOOL	// SPARE
"Q34.7"	Q 34.7	BOOL	// SPARE
"=EU04+EA001-Y0021:1"	Q 35.0	BOOL	// EXTRUDER ZONE 2 COOLING ON
"=EU04+EA001-Y0031:1"	Q 35.1	BOOL	// EXTRUDER ZONE 3 COOLING ON
"=EU04+EA001-Y0041:1"	Q 35.2	BOOL	// EXTRUDER ZONE 4 COOLING ON
"=EU04+EA001-Y0051:1"	Q 35.3	BOOL	// EXTRUDER ZONE 5 COOLING ON
"=EU04+EA001-Y0061:1"	Q 36.0	BOOL	// EXTRUDER ZONE 6 COOLING ON
"=EU04+EA001-Y0071:1"	Q 36.1	BOOL	// EXTRUDER ZONE 7 COOLING ON
"=EU04+EA001-Y0081:1"	Q 36.2	BOOL	// EXTRUDER ZONE 8 COOLING ON
"Q36.3"	Q 36.3	BOOL	// SPARE
"=GI+SK01-1P1:+"	Q 40.0	BOOL	// OPERATING HOURS COUNTER
"=GI+SK01-1K1:A1"	Q 40.1	BOOL	// SIGNAL HORN FAULT INDICATION
"=GI+SK01-2P1:2"	Q 40.2	BOOL	// SIGNAL LAMP RD
"=GI+SK01-2P1:1"	Q 40.3	BOOL	// SIGNAL LAMP YE
"=GI+SK01-2P1:3"	Q 40.4	BOOL	// SPARE
"=GR04+SK01-11Q2:A1"	Q 40.5	BOOL	// PELLETIZER DRIVE MOTOR CONTACTOR ON
"=GR04+SK01-15K2:A1"	Q 40.6	BOOL	// PELLETIZER SAFETY RELAY RESET
"Q40.7"	Q 40.7	BOOL	// SPARE
"Q41.0"	Q 41.0	BOOL	// SPARE
"Q41.1"	Q 41.1	BOOL	// SPARE
"=BE04+SK01-8A1:IN"	Q 41.2	BOOL	// PA013 HEATER PUMP ZONE 2 HEATING ON
"=BE04+PA013-G0102:5"	Q 41.3	BOOL	// PA013 GATE VALVE TO EXTRUDER OPEN
"=BE04+PA013-G0101:5"	Q 41.4	BOOL	// PA013 GATE VALVE RETURN FLOW OPEN
"=GR04+SK01-13K1:RESET"	Q 41.5	BOOL	// PELLETIZER RESET
"=GR04+ZA001-Y0102:1"	Q 41.6	BOOL	// FEED ROLL UP PRESSURE ON
"Q41.7"	Q 41.7	BOOL	// SPARE
"=PS400+SK01-2K1:A1"	Q 42.0	BOOL	// HEATING SUPPLY ON
"+SK01-X4:57"	Q 42.1	BOOL	// SPARE
"Q42.2"	Q 42.2	BOOL	// SPARE
"=EU04+SK01-11T1:16"	Q 42.3	BOOL	// VACUUM PUMP EXTRUDER ON
"Q42.4"	Q 42.4	BOOL	// SPARE
"Q42.5"	Q 42.5	BOOL	// SPARE
"Q42.6"	Q 42.6	BOOL	// SPARE
"=PS400+SK01-2Q1:A1"	Q 42.7	BOOL	// SUPPLY PIPE HEATING ON
"=GR04+SK01-1Q2:A1"	Q 43.0	BOOL	// PUMP WATER BATH ON
"=GR04+SK01-5Q2:A1"	Q 43.1	BOOL	// DRIVE FAN STRAND DEWATERING ON
"=EU04+SK01-7Q2:A1"	Q 43.2	BOOL	// EXTRUDER FREMDBELÜFTUNG START
"=GR04+SK01-21Q2:A1"	Q 43.3	BOOL	// CLASSIFIER VIBRATOR START
"Q43.4"	Q 43.4	BOOL	// SPARE
"Q43.5"	Q 43.5	BOOL	// SPARE
"Q43.6"	Q 43.6	BOOL	// SPARE
"Q43.7"	Q 43.7	BOOL	// SPARE
"TP"	SFB 3	SFB 3	// Generate a Pulse
"TON"	SFB 4	SFB 4	// Generate an On Delay
"TOF"	SFB 5	SFB 5	// Generate an Off Delay
"SET_CLK"	SFC 0	SFC 0	// Set System Clock
"READ_CLK"	SFC 1	SFC 1	// Read System Clock
"DPRD_DAT"	SFC 14	SFC 14	// Read Consistent Data of a Standard DP Slave
"DPWR_DAT"	SFC 15	SFC 15	// Write Consistent Data to a Standard DP Slave
"BLKMOV"	SFC 20	SFC 20	// Copy Variables
"TEST_DB"	SFC 24	SFC 24	// Test Data Block
"RDSYSST"	SFC 51	SFC 51	// Read a System Status List or Partial List
"TIME_TCK"	SFC 64	SFC 64	// Read the System Time
"T_LoadVoltageOnDel_Block"	T 100	TIMER	// Timer: block fault if load voltage is missing
"T_ContVoltageOnDel_Block"	T 101	TIMER	// Timer: block fault if control voltage is missing
"T_DelayFaultCooling_SK01"	T 102	TIMER	// Timer: Delay cooling fault SK01
"T_DelayFaultCooling_CP01"	T 103	TIMER	// Timer: Delay cooling fault CP01
"T_DelayFaultM400SpeedMin"	T 106	TIMER	// Timer: Delay fault M400 Speed Min
"T_DelayFaultP0083_UWL"	T 107	TIMER	// Timer: Delay Upper warning P0083 Vacuum pressure
"T_DelayFaultP0083_UAL"	T 108	TIMER	// Timer: Delay Upper alarm P0083 Vacuum pressure
"T_DelayFaultP0011_LWL"	T 109	TIMER	// Timer: Delay Lower warning P0011 melt pressure
"T_DelayFaultM305_LWL"	T 111	TIMER	// Timer: Delay Lower warning M305 speed
"T_DelayFaultM0001_Ready"	T 112	TIMER	// Timer: Delay Fault Extruder not ready
"T_PA013DelPelletizerOff"	T 116	TIMER	// Timer: Delay Pelletizer off after PA013Stop
"T_DelayFaultF0041_LWL"	T 118	TIMER	// Timer: Delay Lower warning F0041 Nitrogen flow
"T_DelayFaultP0101_LWL"	T 119	TIMER	// Timer: Delay Lower warning P0101 water bath cooling water pressure
"T_DelayG0030"	T 120	TIMER	// Timer: Delay for pelletizer safety door switch
"TimeParameter"	UDT 0	UDT 0	// TimeParameter
"MParameterReal"	UDT 1	UDT 1	// Maschinen Parameter (REAL)
"MParameterDint"	UDT 11	UDT 11	// Maschinen Parameter (DINT)
"BDEParameterREAL"	UDT 101	UDT 101	// BDEParameterREAL
"NomREAL"	UDT 103	UDT 103	// module for nominal value
"ActREAL"	UDT 104	UDT 104	// module for actual value
"MLREAL"	UDT 105	UDT 105	// module for machine level (skaling)
"BDEParameterDINT"	UDT 111	UDT 111	// BDEParameterDINT
"NomDINT"	UDT 113	UDT 113	// module for nominal value
"ActDINT"	UDT 114	UDT 114	// module for actual value
"MLDINT"	UDT 115	UDT 115	// module for machine level
"TContZone"	UDT 427	UDT 427	// heating zone of tcont cp
"EPComSinamicsG120"	UDT 502	UDT 502	// Communication SINAMICS G120
"PIActValueReal"	UDT 1004	UDT 1004	// PIActValueReal
"Graph10Pos"	UDT 1219	UDT 1219	// Visu parameter graph10 positions
"StatesKEY"	UDT 1282	UDT 1282
"EPSlaveDiagDPData"	UDT 1346	UDT 1346	// Slave Diag DP Data
"StatesSEL"	UDT 1397	UDT 1397
"Data ISC-CM Plus H-Type"	UDT 1530	UDT 1530	// Data ISC-CM Plus H-Type
"EPBDH"	UDT 1535	UDT 1535	// Brabender ISC CM plus H-type visualization interface
"ISC-CMp H PConfNom"	UDT 1537	UDT 1537	// brabender ISC CM plus H-type parameter configuration mask for nominal values
"ISC-CMp H PConfAct"	UDT 1538	UDT 1538	// brabender ISC CM plus H-type parameter configuration mask for actual values
"Data KCM LWF-Type"	UDT 1540	UDT 1540	// Data K-Tron Smart K-Link KCM LWF-Type
"EPKDL"	UDT 1545	UDT 1545	// K-Tron dosing controller Smart K-Link KCM / SCM (LWF-Type) visu interface
"KCM LWF PConfNom"	UDT 1547	UDT 1547	// K-Tron Smart K-Link KCM LWF-type parameter configuration mask for nominal values
"KCM LWF PConfAct"	UDT 1548	UDT 1548	// K-Tron Smart K-Link KCM LWF-type parameter configuration mask for actual values
"SkalierungGR01"	VAT 1	
"GR04"	VAT 2	
"General"	VAT 3	
"DB6"	VAT 4	
"EU_Heating"	VAT 5	
"DT04-General"	VAT 6	
"EU_General"	VAT 7	
"VAT_8"	VAT 8	
"KonfigurationDB2"	VAT 10		// KonfigurationDB2
END_SYMBOL_TABLE
